(* IEC 61131-3 sources: SDOHammer4/SDOHammer4.fbsproj/Device.device.xml.v3^/Plc Logic.plclogic.xml.v3^/Application.application.xml.v3^, 2 files *)

(* ---- GVL.gvl ---- *)
(* METADATA
{
	"v3Meta": {
		"objectGuid": "f98b240b-93d2-4c32-bd7d-817c2eb94fac"
	}
}
*)
{attribute 'qualified_only'}
NAMESPACE GVL
// List extracted from MPAStageAlign log files
// by grepping for sdoRead
VAR_GLOBAL CONSTANT
	MAX_VALID_SDOS : INT := 94;
	aValidSDOs : ARRAY[1..MAX_VALID_SDOS] OF STRUCT_SDO_TARGET := [
		( wIndex := 16#1C12, bySubIndex := 1, szSize := XSIZEOF(UINT)),
		( wIndex := 16#1C13, bySubIndex := 1, szSize := XSIZEOF(UINT)),
		( wIndex := 16#2006, bySubIndex := 19, szSize := XSIZEOF(UINT)),
		( wIndex := 16#2050, bySubIndex := 2, szSize := XSIZEOF(DINT)),
		( wIndex := 16#2050, bySubIndex := 2, szSize := XSIZEOF(UDINT)),
		( wIndex := 16#2050, bySubIndex := 3, szSize := XSIZEOF(UDINT)),
		( wIndex := 16#2050, bySubIndex := 4, szSize := XSIZEOF(DINT)),
		( wIndex := 16#2050, bySubIndex := 4, szSize := XSIZEOF(UDINT)),
		( wIndex := 16#2083, bySubIndex := 12, szSize := XSIZEOF(UDINT)),
		( wIndex := 16#2083, bySubIndex := 9, szSize := XSIZEOF(UDINT)),
		( wIndex := 16#2084, bySubIndex := 1, szSize := XSIZEOF(INT)),
		( wIndex := 16#2084, bySubIndex := 29, szSize := XSIZEOF(ULINT)),
		( wIndex := 16#2101, bySubIndex := 15, szSize := XSIZEOF(UINT)),
		( wIndex := 16#2101, bySubIndex := 19, szSize := XSIZEOF(UINT)),
		( wIndex := 16#2101, bySubIndex := 65, szSize := XSIZEOF(UDINT)),
		( wIndex := 16#2102, bySubIndex := 11, szSize := XSIZEOF(UINT)),
		( wIndex := 16#2102, bySubIndex := 12, szSize := XSIZEOF(UINT)),
		( wIndex := 16#2102, bySubIndex := 15, szSize := XSIZEOF(UINT)),
		( wIndex := 16#2102, bySubIndex := 16, szSize := XSIZEOF(UINT)),
		( wIndex := 16#2102, bySubIndex := 19, szSize := XSIZEOF(UINT)),
		( wIndex := 16#2102, bySubIndex := 2, szSize := XSIZEOF(DINT)),
		( wIndex := 16#2102, bySubIndex := 20, szSize := XSIZEOF(UINT)),
		( wIndex := 16#2102, bySubIndex := 21, szSize := XSIZEOF(UINT)),
		( wIndex := 16#2102, bySubIndex := 22, szSize := XSIZEOF(UINT)),
		( wIndex := 16#2102, bySubIndex := 23, szSize := XSIZEOF(UINT)),
		( wIndex := 16#2102, bySubIndex := 24, szSize := XSIZEOF(UINT)),
		( wIndex := 16#2102, bySubIndex := 25, szSize := XSIZEOF(UINT)),
		( wIndex := 16#2102, bySubIndex := 26, szSize := XSIZEOF(UINT)),
		( wIndex := 16#2102, bySubIndex := 27, szSize := XSIZEOF(UINT)),
		( wIndex := 16#2102, bySubIndex := 28, szSize := XSIZEOF(UINT)),
		( wIndex := 16#2102, bySubIndex := 29, szSize := XSIZEOF(UINT)),
		( wIndex := 16#2102, bySubIndex := 30, szSize := XSIZEOF(UINT)),
		( wIndex := 16#2102, bySubIndex := 31, szSize := XSIZEOF(UINT)),
		( wIndex := 16#2102, bySubIndex := 32, szSize := XSIZEOF(UINT)),
		( wIndex := 16#2103, bySubIndex := 10, szSize := XSIZEOF(UINT)),
		( wIndex := 16#2103, bySubIndex := 11, szSize := XSIZEOF(UINT)),
		( wIndex := 16#2103, bySubIndex := 12, szSize := XSIZEOF(UINT)),
		( wIndex := 16#2103, bySubIndex := 13, szSize := XSIZEOF(UINT)),
		( wIndex := 16#2103, bySubIndex := 14, szSize := XSIZEOF(UINT)),
		( wIndex := 16#2103, bySubIndex := 15, szSize := XSIZEOF(UINT)),
		( wIndex := 16#2103, bySubIndex := 5, szSize := XSIZEOF(UINT)),
		( wIndex := 16#2103, bySubIndex := 7, szSize := XSIZEOF(UINT)),
		( wIndex := 16#2103, bySubIndex := 9, szSize := XSIZEOF(UINT)),
		( wIndex := 16#2105, bySubIndex := 10, szSize := XSIZEOF(UINT)),
		( wIndex := 16#2105, bySubIndex := 8, szSize := XSIZEOF(UINT)),
		( wIndex := 16#2106, bySubIndex := 1, szSize := XSIZEOF(UINT)),
		( wIndex := 16#2106, bySubIndex := 10, szSize := XSIZEOF(UINT)),
		( wIndex := 16#2106, bySubIndex := 11, szSize := XSIZEOF(UINT)),
		( wIndex := 16#2106, bySubIndex := 12, szSize := XSIZEOF(UINT)),
		( wIndex := 16#2106, bySubIndex := 13, szSize := XSIZEOF(UINT)),
		( wIndex := 16#2106, bySubIndex := 14, szSize := XSIZEOF(UINT)),
		( wIndex := 16#2106, bySubIndex := 15, szSize := XSIZEOF(UINT)),
		( wIndex := 16#2106, bySubIndex := 2, szSize := XSIZEOF(UINT)),
		( wIndex := 16#2106, bySubIndex := 3, szSize := XSIZEOF(UINT)),
		( wIndex := 16#2106, bySubIndex := 5, szSize := XSIZEOF(UINT)),
		( wIndex := 16#2106, bySubIndex := 6, szSize := XSIZEOF(UINT)),
		( wIndex := 16#2106, bySubIndex := 7, szSize := XSIZEOF(UINT)),
		( wIndex := 16#2106, bySubIndex := 9, szSize := XSIZEOF(UINT)),
		( wIndex := 16#2380, bySubIndex := 1, szSize := XSIZEOF(INT)),
		( wIndex := 16#2380, bySubIndex := 2, szSize := XSIZEOF(INT)),
		( wIndex := 16#2380, bySubIndex := 3, szSize := XSIZEOF(INT)),
		( wIndex := 16#2380, bySubIndex := 4, szSize := XSIZEOF(INT)),
		( wIndex := 16#2500, bySubIndex := 12, szSize := XSIZEOF(INT)),
		( wIndex := 16#2500, bySubIndex := 13, szSize := XSIZEOF(INT)),
		( wIndex := 16#2500, bySubIndex := 14, szSize := XSIZEOF(INT)),
		( wIndex := 16#2500, bySubIndex := 15, szSize := XSIZEOF(INT)),
		( wIndex := 16#2500, bySubIndex := 16, szSize := XSIZEOF(INT)),
		( wIndex := 16#2500, bySubIndex := 17, szSize := XSIZEOF(INT)),
		( wIndex := 16#2500, bySubIndex := 21, szSize := XSIZEOF(UDINT)),
		( wIndex := 16#2500, bySubIndex := 22, szSize := XSIZEOF(UDINT)),
		( wIndex := 16#2500, bySubIndex := 59, szSize := XSIZEOF(DINT)),
		( wIndex := 16#2500, bySubIndex := 61, szSize := XSIZEOF(UDINT)),
		( wIndex := 16#2500, bySubIndex := 66, szSize := XSIZEOF(LINT)),
		( wIndex := 16#2500, bySubIndex := 66, szSize := XSIZEOF(UDINT)),
		( wIndex := 16#2502, bySubIndex := 10, szSize := XSIZEOF(DINT)),
		( wIndex := 16#2502, bySubIndex := 8, szSize := XSIZEOF(DINT)),
		( wIndex := 16#2509, bySubIndex := 12, szSize := XSIZEOF(INT)),
		( wIndex := 16#2514, bySubIndex := 1, szSize := XSIZEOF(UDINT)),
		( wIndex := 16#2514, bySubIndex := 2, szSize := XSIZEOF(UDINT)),
		( wIndex := 16#2514, bySubIndex := 3, szSize := XSIZEOF(UDINT)),
		( wIndex := 16#2514, bySubIndex := 4, szSize := XSIZEOF(UDINT)),
		( wIndex := 16#2514, bySubIndex := 5, szSize := XSIZEOF(DINT)),
		( wIndex := 16#2514, bySubIndex := 6, szSize := XSIZEOF(DINT)),
		( wIndex := 16#2514, bySubIndex := 7, szSize := XSIZEOF(DINT)),
		( wIndex := 16#2514, bySubIndex := 8, szSize := XSIZEOF(DINT)),
		( wIndex := 16#2517, bySubIndex := 1, szSize := XSIZEOF(UDINT)),
		( wIndex := 16#6060, bySubIndex := 0, szSize := XSIZEOF(INT)),
		( wIndex := 16#6096, bySubIndex := 1, szSize := XSIZEOF(UDINT)),
		( wIndex := 16#6096, bySubIndex := 2, szSize := XSIZEOF(UDINT)),
		( wIndex := 16#6097, bySubIndex := 1, szSize := XSIZEOF(UDINT)),
		( wIndex := 16#6097, bySubIndex := 2, szSize := XSIZEOF(UDINT)),
		( wIndex := 16#60A2, bySubIndex := 1, szSize := XSIZEOF(UDINT)),
		( wIndex := 16#60A2, bySubIndex := 2, szSize := XSIZEOF(UDINT)),
		( wIndex := 16#6123, bySubIndex := 0, szSize := XSIZEOF(ULINT))
	];
END_VAR

END_NAMESPACE

(* ---- PLC_PRG.prg.st ---- *)
(* METADATA
{
	"v3Meta": {
		"objectGuid": "265bd9e0-f119-4664-b8ae-ea3439835427"
	}
}
*)
PROGRAM PLC_PRG
VAR
    // Array of independent function blocks for parallel execution
    aSdoReaders     : ARRAY[1..4] OF ETC_CO_SdoRead;

    // Independent states for each slave's execution loop
    aStates         : ARRAY[1..4] OF INT := [4(0)];

    // Configuration for 4 slaves (Populate with actual Node IDs from your device tree)
    aSlaveIds       : ARRAY[1..4] OF UINT;
    SlaveCount      : INT := 0;

    // Unique data buffers and random parameters per slave pipeline
    aDataBuffs      : ARRAY[1..4] OF ARRAY[0..255] OF BYTE;
    aRandIndices    : ARRAY[1..4] OF WORD;
    aRandSubIndices : ARRAY[1..4] OF BYTE;
    aRandSizes      : ARRAY[1..4] OF CAA.SIZE;

    // Shared seed for the pseudo-random number generator
    dwRandSeed      : DWORD := 987654321;

    // Performance Metrics
    aReadCounts     : ARRAY[1..4] OF UDINT;
    aErrorCounts    : ARRAY[1..4] OF UDINT;
	aLastErrorCodes : ARRAY[1..4] OF ETC_CO_ERROR;
    aLastAbortCodes : ARRAY[1..4] OF DWORD;
    aReadStartTime  : ARRAY[1..4] OF SYSTIME;
    aReadEndTime    : ARRAY[1..4] OF SYSTIME;
    aElapsed        : ARRAY[1..4] OF ULINT;
	aTotalElapsed   : ARRAY[1..4] OF ULINT;
    aAverageTime    : ARRAY[1..4] OF REAL;

    // Iterator loop index
    i               : INT;

    // Pointer to traverse the sequential linked list
    pSlave          : POINTER TO ETCSlave;

	udiTargetIndex  : UDINT;

    bInitialized    : BOOL := FALSE;

	lastCycleTime   : SYSTIME;
	thisCycleTime   : SYSTIME;
	cycleTime       : SYSTIME;

END_VAR

IF NOT bInitialized THEN

	// wait for all slaves to be identified and linked into a list
	IF NOT EtherCAT_Master.xConfigFinished THEN
	    SlaveCount := 0;
		RETURN;
	END_IF

    // Fetch the entry point of the linked list from the Master node
    // Replace 'EtherCAT_Master' with the exact name of your master node
	IF 0 = pSlave THEN
		pSlave := EtherCAT_Master.FirstSlave;
	END_IF

	IF 0 = pSlave THEN
		// end of list, we're ready
		bInitialized := TRUE;
		RETURN;
	END_IF

	// wait for addresses to be assigned
	IF 0 = pSlave^.PhysSlaveAddr THEN
		RETURN;
	END_IF

	// got an address, advance to next one for next bus cycle
	SlaveCount := SlaveCount + 1;
	aSlaveIds[SlaveCount] := pSlave^.PhysSlaveAddr;
	IF 4 = SlaveCount THEN
		bInitialized := TRUE; // no more space, so start
	ELSE
		pSlave := pSlave^.NextInstance;
		RETURN;
	END_IF

END_IF

SysTimeGetUs(thisCycleTime);
cycleTime := thisCycleTime - lastCycleTime;
lastCycleTime := thisCycleTime;

// Loop through and evaluate all 4 state machines independently in the same PLC cycle
FOR i := 1 TO SlaveCount DO

    CASE aStates[i] OF
        0: // GENERATE PARAMETERS & PREPARE
            // Step the shared LCG pseudo-random generator
            dwRandSeed := (dwRandSeed * 1103515245 + 12345) MOD 16#7FFFFFFF;

			// Map the random value bounded strictly to your extracted ESI array length
			udiTargetIndex := TO_UDINT((dwRandSeed MOD TO_DWORD(GVL.MAX_VALID_SDOS)) + 1);

			// Pull valid paired parameters cleanly
			aRandIndices[i]    := GVL.aValidSDOs[udiTargetIndex].wIndex;
			aRandSubIndices[i] := GVL.aValidSDOs[udiTargetIndex].bySubIndex;
			aRandSizes[i]      := GVL.aValidSDOs[udiTargetIndex].szSize;

			// Reset the FB execute trigger
			aSdoReaders[i](xExecute := FALSE);
			SysTimeGetUs(aReadStartTime[i]);
			aStates[i] := 1;

        1: // TRIGGER & MONITOR READS IN PARALLEL
            aSdoReaders[i](
                xExecute    := TRUE,
                usiCom      := 1,
                uiDevice    := aSlaveIds[i],
                wIndex      := aRandIndices[i],
                bySubindex  := aRandSubIndices[i],
                pBuffer     := ADR(aDataBuffs[i]),
                szSize      := aRandSizes[i],
                udiTimeOut  := 10
            );

            IF aSdoReaders[i].xDone THEN
                aReadCounts[i] := aReadCounts[i] + 1;
				ComputeTime();
                aSdoReaders[i](xExecute := FALSE);
                aStates[i] := 0; // Instantly queue the next read

            ELSIF aSdoReaders[i].xError THEN
                aReadCounts[i] := aReadCounts[i] + 1;
				ComputeTime();
                aErrorCounts[i] := aErrorCounts[i] + 1;
				aLastErrorCodes[i] := aSdoReaders[i].eError;
                aLastAbortCodes[i] := aSdoReaders[i].udiSdoAbort;
                aSdoReaders[i](xExecute := FALSE);
                aStates[i] := 0; // Skip error and keep hammering
            END_IF

    END_CASE

END_FOR
END_PROGRAM
